// TIA Portal V17 export
// export: Created 2024-09-02T12:49:57.217454Z, ExportSetting WithDefaults, DisplayName Totally Integrated Automation Portal, DisplayVersion V17, DisplayName TIA Portal Openness, DisplayVersion V17, DisplayName TIA Portal Version Control Interface, DisplayVersion V17, DisplayName STEP 7 Professional, DisplayVersion V17, DisplayName STEP 7 Safety, DisplayVersion V17, DisplayName WinCC Professional, DisplayVersion V17
FUNCTION "HLP_BooltoByte" : Void   // FC30001, LAD
TITLE = Transfer Bool to Byte
{ S7_Optimized_Access := 'TRUE' }
AUTHOR : O.Fuehrus
FAMILY : HLP
NAME : HLP
VERSION : 1.0
// stored: AutoNumber false, IsIECCheckEnabled false, SetENOAutomatically false, UDAEnableTagReadback false
   VAR_INPUT
      IN0 : Bool;
      IN1 : Bool;
      IN2 : Bool;
      IN3 : Bool;
      IN4 : Bool;
      IN5 : Bool;
      IN6 : Bool;
      IN7 : Bool;
   END_VAR
   VAR_OUTPUT
      oByte : Byte;
   END_VAR
BEGIN

REGION Network 1: Bits
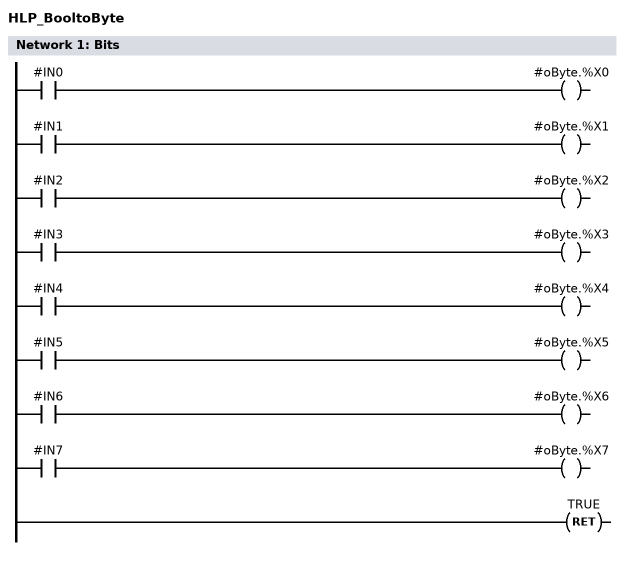
   RUNG wire#powerrail
      Contact( #IN0 )
      Coil( #oByte.%X0 )
   END_RUNG
   RUNG wire#powerrail
      Contact( #IN1 )
      Coil( #oByte.%X1 )
   END_RUNG
   RUNG wire#powerrail
      Contact( #IN2 )
      Coil( #oByte.%X2 )
   END_RUNG
   RUNG wire#powerrail
      Contact( #IN3 )
      Coil( #oByte.%X3 )
   END_RUNG
   RUNG wire#powerrail
      Contact( #IN4 )
      Coil( #oByte.%X4 )
   END_RUNG
   RUNG wire#powerrail
      Contact( #IN5 )
      Coil( #oByte.%X5 )
   END_RUNG
   RUNG wire#powerrail
      Contact( #IN6 )
      Coil( #oByte.%X6 )
   END_RUNG
   RUNG wire#powerrail
      Contact( #IN7 )
      Coil( #oByte.%X7 )
   END_RUNG
   RUNG wire#powerrail
      ReturnCoil( TRUE )
   END_RUNG
   // the same network as SCL:
   #oByte.%X0 := #IN0;
   #oByte.%X1 := #IN1;
   #oByte.%X2 := #IN2;
   #oByte.%X3 := #IN3;
   #oByte.%X4 := #IN4;
   #oByte.%X5 := #IN5;
   #oByte.%X6 := #IN6;
   #oByte.%X7 := #IN7;
   ENO := TRUE;
   RETURN;
END_REGION
END_FUNCTION
